// Mitsubishi GX Works2 project: ProjectBb   PLC: FX3G

// global labels: Global1
VAR_GLOBAL
  StartMachine AT X010 : BOOL;
  MachineWorking AT Y001 : BOOL;
  StopMachine AT M0 : BOOL;
  CarInPlace AT X001 : BOOL;
  startblinking AT M1 : BOOL;
  Temp2 AT M2 : BOOL;
  Temp3 AT M3 : BOOL;
  Timer1 AT TC1 : BOOL;
END_VAR
VAR_GLOBAL CONSTANT
  Timer10 : INT := 10;
END_VAR
VAR_GLOBAL
  TimerFinished1 AT TS1 : BOOL;
  Lamp0 AT M4 : BOOL;
  Timer2 AT TC2 : BOOL;
  TimerFinished2 AT TS2 : BOOL;
  Lamp1 AT M5 : BOOL;
  TimerMoving AT TC3 : BOOL;
END_VAR
VAR_GLOBAL CONSTANT
  Timer40 : INT := 40;
END_VAR
VAR_GLOBAL
  TimerFinished3 AT TS3 : BOOL;
  Lamp01 AT Y003 : BOOL;
  CarInWashingPlace AT X002 : BOOL;
  AnalogInput2 AT D8281 : INT;
END_VAR
VAR_GLOBAL CONSTANT
  Ten : REAL := 10;
  Min20 : REAL := 20;
  Max50 : REAL := 50;
END_VAR
VAR_GLOBAL
  GoodPreasure1 AT M10 : BOOL;
  GoodPreasure2 AT M11 : BOOL;
  PreasureIsOk AT M12 : BOOL;
  TimerWashing AT TC5 : BOOL;
  TimerFinished5 AT TS5 : BOOL;
  WashingFinished AT M13 : BOOL;
  TimerSoap AT TC6 : BOOL;
END_VAR
VAR_GLOBAL CONSTANT
  Timer20 : INT := 20;
END_VAR
VAR_GLOBAL
  TimerFinished6 AT TS6 : BOOL;
  Soap AT Y005 : BOOL;
  WashingFinished2 AT Y004 : BOOL;
  PresureUnder50 AT X004 : BOOL;
  PresureUnder20 AT X003 : BOOL;
  PresureNotOk AT Y002 : BOOL;
  CounterWashing AT CC1 : BOOL;
END_VAR
VAR_GLOBAL CONSTANT
  Four : INT := 4;
END_VAR
VAR_GLOBAL
  WashingFinished3 AT CS1 : BOOL;
  Error AT X005 : BOOL;
  CarInWashingPlace2 AT X006 : BOOL;
  CounterWashing2 AT CC2 : BOOL;
  WashingFinished4 AT CS2 : BOOL;
END_VAR
VAR_GLOBAL CONSTANT
  Two : INT := 2;
  Timer50 : INT := 50;
END_VAR
VAR_GLOBAL
  CounterBlinking AT CC2 : BOOL;
END_VAR
VAR_GLOBAL CONSTANT
  One : INT := 1;
END_VAR
VAR_GLOBAL
  Temp1 AT M200 : BOOL;
  CounterBlinkingFinished AT CS2 : BOOL;
END_VAR

// task Task_01 (event TRUE, interval 0, priority 31): POU_01

PROGRAM POU_01
(* structured ladder/FBD written out as ST: instructions are called as NAME(EN, inputs, outputs); _pN, _eN, _tN stand for wires *)
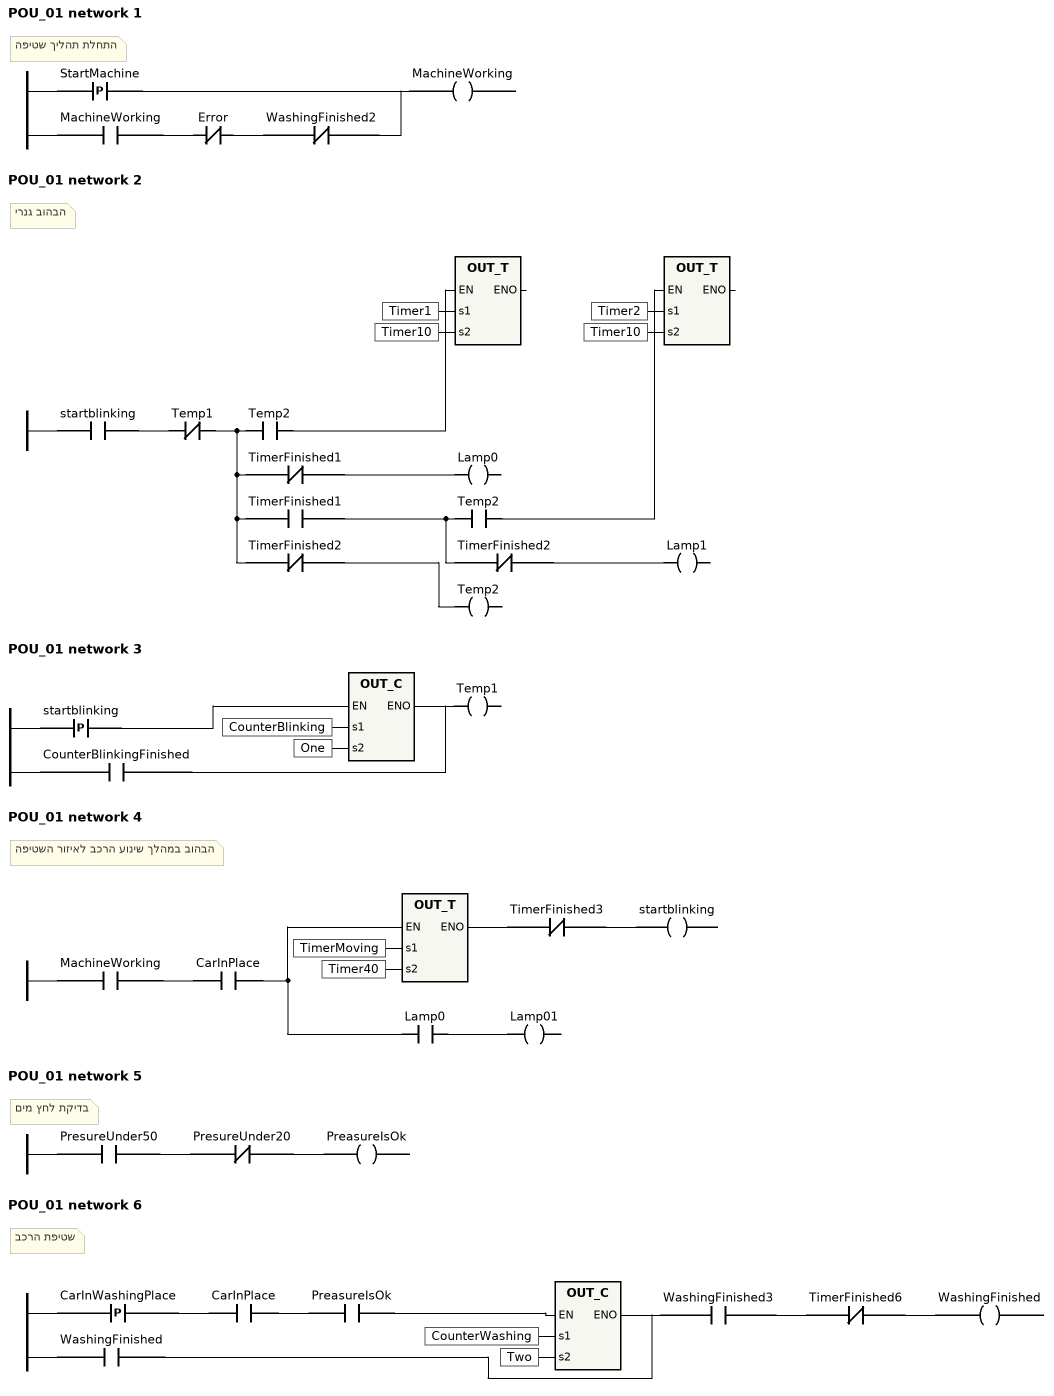
(* network 1 *)
(* התחלת תהליך שטיפה *)
MachineWorking := LDP(TRUE, StartMachine) OR (MachineWorking AND NOT Error AND NOT WashingFinished2);
(* network 2 *)
(* הבהוב גנרי *)
_p1 := startblinking AND NOT Temp1;
OUT_T(_p1 AND Temp2, Timer1, Timer10);
Lamp0 := _p1 AND NOT TimerFinished1;
_p2 := _p1 AND TimerFinished1;
OUT_T(_p2 AND Temp2, Timer2, Timer10);
Lamp1 := _p2 AND NOT TimerFinished2;
Temp2 := _p1 AND NOT TimerFinished2;
(* network 3 *)
_e1 := OUT_C(LDP(TRUE, startblinking), CounterBlinking, One);
Temp1 := _e1 OR CounterBlinkingFinished;
(* network 4 *)
(* הבהוב במהלך שינוע הרכב לאיזור השטיפה *)
_p1 := MachineWorking AND CarInPlace;
_e2 := OUT_T(_p1, TimerMoving, Timer40);
startblinking := _e2 AND NOT TimerFinished3;
Lamp01 := _p1 AND Lamp0;
(* network 5 *)
(* בדיקת לחץ מים *)
PreasureIsOk := PresureUnder50 AND NOT PresureUnder20;
(* network 6 *)
(* שטיפת הרכב *)
_e1 := OUT_C(LDP(TRUE, CarInWashingPlace) AND CarInPlace AND PreasureIsOk, CounterWashing, Two);
WashingFinished := ((_e1 OR WashingFinished) AND WashingFinished3) AND NOT TimerFinished6;
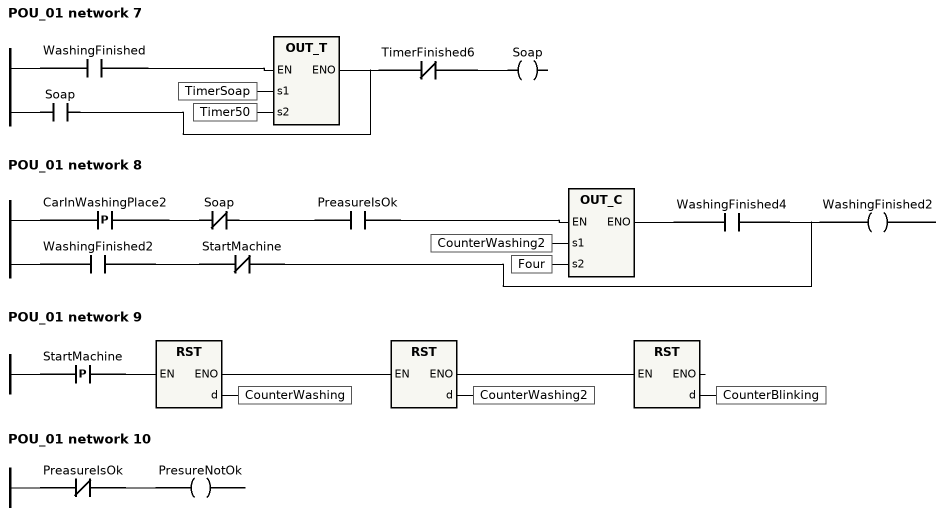
(* network 7 *)
_e1 := OUT_T(WashingFinished, TimerSoap, Timer50);
Soap := (_e1 OR Soap) AND NOT TimerFinished6;
(* network 8 *)
_e1 := OUT_C(LDP(TRUE, CarInWashingPlace2) AND NOT Soap AND PreasureIsOk, CounterWashing2, Four);
WashingFinished2 := (_e1 AND WashingFinished4) OR (WashingFinished2 AND NOT StartMachine);
(* network 9 *)
_e1 := RST(LDP(TRUE, StartMachine), CounterWashing);
_e2 := RST(_e1, CounterWashing2);
RST(_e2, CounterBlinking);
(* network 10 *)
PresureNotOk := NOT PreasureIsOk;
END_PROGRAM
